GLOBALCONSTANTS Industry_Groups (* ISOBUS Industry Group defines *)
  (* Standard: 61499-1 *)
  (* Version 1.0, 2026-06-29, Franz Höpfinger, Demmler Andreas Fahrzeugbau *)
  PACKAGE isobus::pgn::const;
  VAR_GLOBAL CONSTANT
    IG_GLOBAL : BYTE := 0; (* Industry Group: Global, applies to all *)
    IG_ON_HIGHWAY_EQUIPMENT : BYTE := 1; (* Industry Group: On-Highway Equipment *)
    IG_AGRICULTURAL_AND_FORESTRY_EQUIPMENT : BYTE := 2; (* Industry Group: Agricultural and Forestry Equipment *)
    IG_CONSTRUCTION_EQUIPMENT : BYTE := 3; (* Industry Group: Construction Equipment *)
    IG_MARINE : BYTE := 4; (* Industry Group: Marine *)
    IG_INDUSTRIAL_PROCESS_CONTROL_STATIONARY : BYTE := 5; (* Industry Group: Industrial-Process Control-Stationary (Gen-Sets) *)
    IG_RESERVED_FOR_FUTURE_ASSIGNMENT_BY_SAE : BYTE := 6; (* Industry Group: Reserved for future assignment by SAE *)
    IG_RESERVED_FOR_FUTURE_ASSIGNMENT_BY_SAE_7 : BYTE := 7; (* Industry Group: Reserved for future assignment by SAE *)
  END_VAR
END_GLOBALCONSTANTS
